Yaskawa INFORM job: R2_W53-A1(90,180)AWOK.JBI

/JOB
//NAME R2_W53-A1(90,180)AWOK
///FOLDERNAME AWOK
//POS
///NPOS 36,36,0,2,0,0
///TOOL 0
///POSTYPE PULSE
///PULSE
C00000=29586,64241,-25483,43781,98921,43724
C00001=57127,76182,10095,53684,99903,33351
C00002=68868,95750,33777,40131,101998,35545
C00003=80579,136048,88691,13195,105824,34209
C00004=80579,135466,89528,13135,105030,34121
C00005=80614,135877,90680,13103,104541,34078
C00006=80579,135466,89528,13135,105030,34121
C00007=80098,138136,91616,11040,112385,45139
C00008=80579,134296,92856,2574,121038,58729
C00009=80445,131950,90268,2542,121430,58686
C00010=80579,134296,92856,2574,121038,58729
C00011=78176,133439,87120,21461,107379,43183
C00012=80582,134264,97775,32660,78294,14244
C00013=80553,132262,95759,32645,78486,14287
C00014=80580,135158,102153,32903,76401,13683
C00015=80506,135744,102968,32942,76262,13611
C00016=80580,135158,102153,32903,76401,13683
C00017=79366,137379,99712,32902,79107,13996
C00018=76874,109703,51513,11024,106473,-11901
C00019=80591,100267,38822,2686,105144,-12380
C00020=80592,98128,39662,2663,103530,-12415
C00021=80278,98755,41840,2698,102520,-12539
C00022=80323,95098,37876,2698,103081,-12510
C00023=80415,96751,38231,2692,103708,-12467
C00024=79496,98741,42532,-2001,99764,-12323
C00025=80580,97640,39756,-2642,100727,-11961
C00026=80580,99717,38880,-2660,102332,-11996
C00027=78782,132344,81667,13923,102302,-75965
C00028=82527,146785,106393,12485,99041,-75185
C00029=79289,148877,112583,13562,98534,-76260
C00030=76253,124275,81193,14214,102523,-76798
C00031=76429,114978,64746,14154,104138,-76557
C00032=76429,114978,64746,14154,104138,-76557
C00033=76429,128622,61528,15029,112853,-75461
C00034=76429,128622,61528,15029,59041,-75461
C00035=50666,136252,61528,15029,59041,-75461
BC00000=15470,258107,1075171
BC00001=15470,185409,1075171
BC00002=15470,185409,1075171
BC00003=15469,185409,1075175
BC00004=15999,185447,1075175
BC00005=15992,184880,1075175
BC00006=15999,185447,1075175
BC00007=17464,163759,1075175
BC00008=19492,133752,1075175
BC00009=19488,135596,1075175
BC00010=19492,133752,1075175
BC00011=20512,176597,1075175
BC00012=21980,238233,1075175
BC00013=21994,241675,1075175
BC00014=21994,241675,1075175
BC00015=23686,241671,1075175
BC00016=21994,241675,1075175
BC00017=21994,241675,1075175
BC00018=871,188297,1075175
BC00019=871,188297,1075175
BC00020=1360,184158,1075175
BC00021=1421,183643,1075175
BC00022=1555,182503,1075175
BC00023=1555,182503,1075175
BC00024=26602,181892,1075175
BC00025=28340,183369,1075175
BC00026=27012,187457,1075175
BC00027=26690,187409,1075175
BC00028=26690,187409,1075175
BC00029=26690,187409,1075175
BC00030=26690,187409,1075175
BC00031=26690,187409,1075175
BC00032=26690,187409,1075175
BC00033=26690,187409,1075175
BC00034=26690,267974,1075175
BC00035=26690,436009,1075175
///POSTYPE BASE
///RECTAN
///RCONF 0,0,0,0,0,0,0,0,0,0,0,0,0,0,0,0,0,0,0,0,0,0,0,0
P00006=0.222,-3.123,-1.508,0.0000,0.0000,0.0000
P00022=0.222,-3.123,-1.508,0.0000,0.0000,0.0000
//INST
///DATE 2023/11/16 17:53
///ATTR SC,RW
///GROUP1 RB1,BS1
NOP
'r2_W53-A1(90,180)
'Path S1056
SFTOF
MOVJ C00000 BC00000 VJ=20.00
MOVJ C00001 BC00001 VJ=20.00
MOVJ C00002 BC00002 VJ=20.00
MOVL C00003 BC00003 V=100.0
MOVL C00004 BC00004 V=60.0
REFP 3 C00005 BC00005
CALL JOB:SEARCH-R1
SET P022 P006
SFTON P022
MOVL C00006 BC00006 V=60.0
MOVL C00007 BC00007 V=60.0
MOVL C00008 BC00008 V=60.0
REFP 3 C00009 BC00009
CALL JOB:SEARCH-R1
SET P022 P006
SFTON P022
MOVL C00010 BC00010 V=60.0
MOVL C00011 BC00011 V=60.0
MOVL C00012 BC00012 V=100.0
MOVL C00013 BC00013 V=60.0
MOVL C00014 BC00014 V=60.0
REFP 3 C00015 BC00015
CALL JOB:SEARCH-R1
SET P022 P006
SFTON P022
MOVL C00016 BC00016 V=60.0
MOVL C00017 BC00017 V=100.0
'Path W1057
SFTOF
SFTON P022
MOVJ C00018 BC00018 VJ=20.00
MOVJ C00019 BC00019 VJ=20.00 PL=0
MOVL C00020 BC00020 V=100.0
MOVL C00021 BC00021 V=100.0 PL=0
REFP 1 C00022 BC00022
REFP 2 C00023 BC00023
MACRO1 MJ#(0) ARGF6
ARCON
MOVL C00024 BC00024 V=11.7
ARCOF
MOVL C00025 BC00025 V=100.0
MOVL C00026 BC00026 V=100.0
SFTOF
SFTON P022
'COMMENT
MOVJ C00027 BC00027 VJ=20.00
MOVL C00028 BC00028 V=100.0 PL=0
MACRO1 MJ#(0) ARGF6
ARCON
MOVL C00029 BC00029 V=11.7
MOVL C00030 BC00030 V=11.7
ARCOF
MOVL C00031 BC00031 V=100.0
MOVL C00032 BC00032 V=100.0
MOVJ C00033 BC00033 VJ=20.00
MOVJ C00034 BC00034 VJ=20.00
SFTOF
MOVJ C00035 BC00035 VJ=20.00
END
